{attribute 'qualified_only'}
{attribute 'strict'}
TYPE eSERVICE :
(
	Backup			:=0,
	Backup_RevDocu	:=1,
	Restore			:=2

);
END_TYPE

(* stored: Version 1.1.0.1, ProductVersion 3.1.4024.6
   EnumerationTextList eSERVICE: Id {ea8750c0-faca-4d6a-873d-642b55d011d4} *)
